// TIA Portal V19 export
DATA_BLOCK "IEC_Timer_0_DB_83"   // DB144
{ S7_Optimized_Access := 'TRUE' }
// stored: InstanceOfName IEC_TIMER, OfSystemLibElement IEC_TIMER, OfSystemLibVersion 1.0
"IEC_TIMER"
   // VAR
   //    PT : Time;
   //    ET { ExternalWritable := 'False'} : Time;
   //    IN : Bool;
   //    Q { ExternalWritable := 'False'} : Bool;
   // END_VAR
BEGIN
END_DATA_BLOCK
